# B&R Automation Studio project CoffeeMachine
Automation Studio 4.12.9.18 SP; Default project; technology packages: Acp10Arnc0 5.16.2

## Configuration PP65mcSim

CPU 4PP065.0571-P74, AutomationRuntime E3.10, Build 4.1.2, Safety 0.0, Vc V4.72.6

### Task classes (Cpu.sw)
```
Cyclic#1 (cycle 10000 us, tolerance 10000 us):
  mainlogic <- mainlogic.prg
  feeder <- FeederArm.feeder.prg
  conveyor <- ConveyorBelt.conveyor.prg
  brewing <- BrewingAssembly.brewing.prg
  heating <- FlowHeater.heating.prg
Cyclic#4 (cycle 100000 us, tolerance 100000 us):
  visCtrl <- Visualisation.visCtrl.prg
  visAlarm <- Visualisation.visAlarm.prg
  visTrend <- Visualisation.visTrend.prg
DataObjects: cappu <- Recipes.cappu.dob, regular <- Recipes.regular.dob, espres <- Recipes.espres.dob, Acp10sys
NcDataObjects: acp_err <- FeederArm.acp_err.dob, motor_sim <- FeederArm.motor_sim.dob, motor_offi <- FeederArm.motor_office.dob, feed_ini <- FeederArm.feed_ini.dob, conv_ini <- ConveyorBelt.conv_ini.dob
Binaries: vccalarm, vcclbox, vcctext, vcrt, VisuW03, vccnum, vcchspot, vccbar, vccurl, vcchtml, vcfile, arialxsr, vcpdsw, vccbmp, vcshared, vcctrend, vcfntttf, vcgclass, vccovl, arialbd, vcdsint, vccslider, vcalarm, vccline, vcresman, vcdsloc, vccbtn, vccstr, vcbclass, vcxml, VisuW02, arial, vccdt, vccgauge, vccshape, arconfig, sysconf, ashwd, asfw, iomap, Acp10map, Acp10cfg, vctcal, vcpfmtcx, vcpdi815, VisuW01, visvc, vcpdi855, vcpfpp50, vcpdihd, vcptelo, vcmgr
Libraries: Acp10sdc, standard, loopconr, astime, runtime, powerlnk, CoffeeLib, Acp10par, AsArSdm, NcGlobal, brsystem, sys_lib, Acp10man, fileio, dataobj, acp10_mc, visapi
```

### Hardware
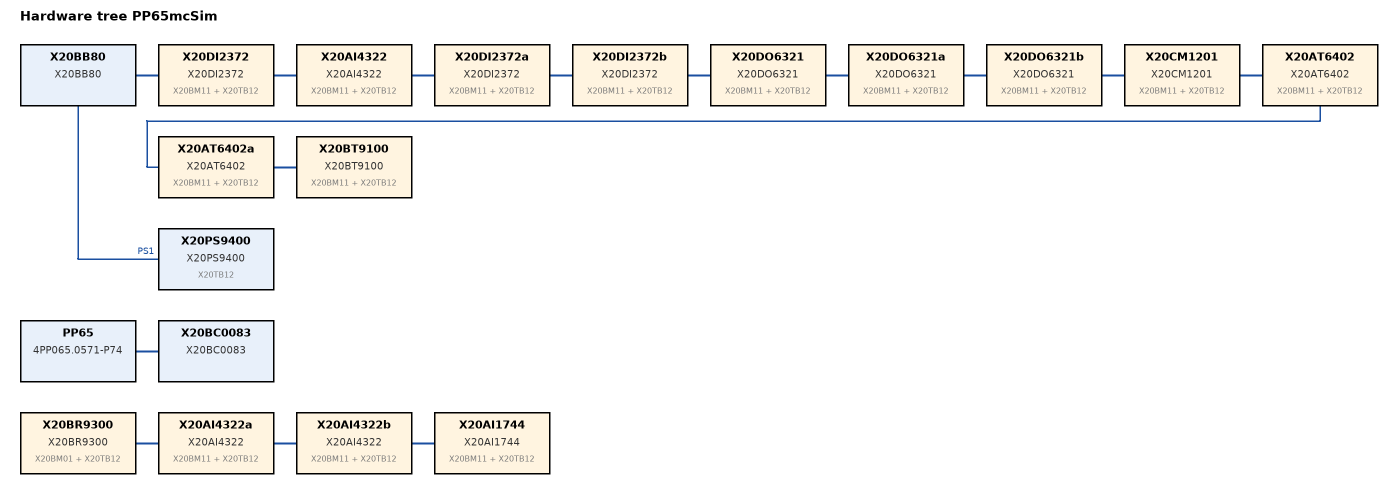
```
PP65 : 4PP065.0571-P74 v1.2.0.0
  Connector IF4:
    DNAConfiguration = manual
  Connector IF5:
    ActivateDevice = 1
    HostName = pp500coffeemachine
    Mode = Manual
    InternetAddress = 10.49.40.222
    SubnetMask = 255.255.255.0
  PreserveNonVolatileSystemSettings = 0
  BRObjects = 450
  Cyclic1Duration = 10000
  Cyclic1Tolerance = 10000
  Cyclic2Duration = 20000
  Cyclic2Tolerance = 20000
  Cyclic3Duration = 50000
  Cyclic3Tolerance = 50000
  Cyclic4Duration = 100000
  Cyclic4Tolerance = 100000
  Cyclic5Duration = 200000
  Cyclic5Tolerance = 200000
  Cyclic6Duration = 500000
  Cyclic6Tolerance = 500000
  Cyclic7Duration = 1000000
  Cyclic7Tolerance = 1000000
  Cyclic8Duration = 10000
  Cyclic8Tolerance = 30000000
  EthernetHostName = brautomation
  ActivateDns = 1
X20AI1744 : X20AI1744 v1.10.0.0  [SS1 -> X20TB12o.SS; SL -> X20BM11m.SL1]
  Supervision = off
X20AI4322 : X20AI4322 v1.2.0.0  [SS1 -> X20TB12b.SS; SL -> X20BM11a.SL1]
  Supervision = off
X20AI4322a : X20AI4322 v1.2.0.0  [SS1 -> X20TB12m.SS; SL -> X20BM11k.SL1]
  Supervision = off
X20AI4322b : X20AI4322 v1.2.0.0  [SS1 -> X20TB12n.SS; SL -> X20BM11l.SL1]
  Supervision = off
X20AT6402 : X20AT6402 v1.2.0.0  [SS1 -> X20TB12i.SS; SL -> X20BM11h.SL1]
  Supervision = off
X20AT6402a : X20AT6402 v1.2.0.0  [SS1 -> X20TB12j.SS; SL -> X20BM11i.SL1]
  Supervision = off
X20BB80 : X20BB80 v1.1.0.0
X20BC0083 : X20BC0083 v2.16.0.0  [PLK1 -> PP65.IF4 (NodeNumber=1) [Cable Type=PowerlinkCable, Length=10, Version=1.0.0.3]; SL -> X20BB80.SL1]
  Supervision = off
X20BM01 : X20BM01 v2.2.0.0
X20BM11 : X20BM11 v1.1.0.0  [X2X1 -> X20BB80.IF1]
X20BM11a : X20BM11 v1.1.0.0  [X2X1 -> X20BM11.X2X2]
X20BM11b : X20BM11 v1.1.0.0  [X2X1 -> X20BM11a.X2X2]
X20BM11c : X20BM11 v1.1.0.0  [X2X1 -> X20BM11b.X2X2]
X20BM11d : X20BM11 v1.1.0.0  [X2X1 -> X20BM11c.X2X2]
X20BM11e : X20BM11 v1.1.0.0  [X2X1 -> X20BM11d.X2X2]
X20BM11f : X20BM11 v1.1.0.0  [X2X1 -> X20BM11e.X2X2]
X20BM11g : X20BM11 v1.1.0.0  [X2X1 -> X20BM11f.X2X2]
X20BM11h : X20BM11 v1.1.0.0  [X2X1 -> X20BM11g.X2X2]
X20BM11i : X20BM11 v1.1.0.0  [X2X1 -> X20BM11h.X2X2]
X20BM11j : X20BM11 v1.1.0.0  [X2X1 -> X20BM11i.X2X2]
X20BM11k : X20BM11 v1.1.0.0  [X2X1 -> X20BM01.X2X2]
X20BM11l : X20BM11 v1.1.0.0  [X2X1 -> X20BM11k.X2X2]
X20BM11m : X20BM11 v1.1.0.0  [X2X1 -> X20BM11l.X2X2]
X20BR9300 : X20BR9300 v1.3.0.0  [SS1 -> X20TB12l.SS; SL -> X20BM01.SL1; X2X1 -> X20BT9100.X2X1 [Cable Type=X2XCable, Length=10, Version=1.0.0.3]]
  Supervision = off
X20BT9100 : X20BT9100 v1.3.0.0  [SS1 -> X20TB12k.SS; SL -> X20BM11j.SL1]
  Supervision = off
X20CM1201 : X20CM1201 v1.2.0.0  [SS1 -> X20TB12h.SS; SL -> X20BM11g.SL1]
  Supervision = off
X20DI2372 : X20DI2372 v1.2.0.0  [SS1 -> X20TB12a.SS; SL -> X20BM11.SL1]
  Supervision = off
X20DI2372a : X20DI2372 v1.2.0.0  [SS1 -> X20TB12c.SS; SL -> X20BM11b.SL1]
  Supervision = off
X20DI2372b : X20DI2372 v1.2.0.0  [SS1 -> X20TB12d.SS; SL -> X20BM11c.SL1]
  Supervision = off
X20DO6321 : X20DO6321 v1.2.0.0  [SS1 -> X20TB12e.SS; SL -> X20BM11d.SL1]
  Supervision = off
X20DO6321a : X20DO6321 v1.2.0.0  [SS1 -> X20TB12f.SS; SL -> X20BM11e.SL1]
  Supervision = off
X20DO6321b : X20DO6321 v1.2.0.0  [SS1 -> X20TB12g.SS; SL -> X20BM11f.SL1]
  Supervision = off
X20PS9400 : X20PS9400 v1.8.0.0  [SS1 -> X20TB12.SS; PS -> X20BB80.PS1]
  Supervision = off
X20TB12 : X20TB12 v1.0.0.0
X20TB12a : X20TB12 v1.0.0.0
X20TB12b : X20TB12 v1.0.0.0
X20TB12c : X20TB12 v1.0.0.0
X20TB12d : X20TB12 v1.0.0.0
X20TB12e : X20TB12 v1.0.0.0
X20TB12f : X20TB12 v1.0.0.0
X20TB12g : X20TB12 v1.0.0.0
X20TB12h : X20TB12 v1.0.0.0
X20TB12i : X20TB12 v1.0.0.0
X20TB12j : X20TB12 v1.0.0.0
X20TB12k : X20TB12 v1.0.0.0
X20TB12l : X20TB12 v1.0.0.0
X20TB12m : X20TB12 v1.0.0.0
X20TB12n : X20TB12 v1.0.0.0
X20TB12o : X20TB12 v1.0.0.0
```

## Configuration Simulation

CPU , AutomationRuntime I4.93, Build 4.1.2, Safety 0.0, Vc V4.73.3

### Task classes (AppMo.sw)
```
Cyclic#1 (cycle 10000 us, tolerance 0 us):
  myApptask1 <- myAppMod1.myApptask1.prg
```

### Task classes (Cpu.sw)
```
Cyclic#1 (cycle 10000 us, tolerance 0 us):
  mainlogic <- mainlogic.prg
  feeder <- FeederArm.feeder.prg
  conveyor <- ConveyorBelt.conveyor.prg
  brewing <- BrewingAssembly.brewing.prg
  heating <- FlowHeater.heating.prg
Cyclic#2:
  visCtrl <- Visualisation.visCtrl.prg
Cyclic#4:
  visAlarm <- Visualisation.visAlarm.prg
  visTrend <- Visualisation.visTrend.prg
  myProg <- myProg.prg
DataObjects: regular <- Recipes.regular.dob, cappu <- Recipes.cappu.dob, espres <- Recipes.espres.dob, empty1 <- Recipes.empty1.dob, object2 <- Recipes.object2.dob, data <- data.dob
NcDataObjects: acp_err <- FeederArm.acp_err.dob, motor_sim <- FeederArm.motor_sim.dob, motor_offi <- FeederArm.motor_office.dob, feed_ini <- FeederArm.feed_ini.dob, conv_ini <- ConveyorBelt.conv_ini.dob, cnc1 <- cnc1.dob, cnc2 <- cnc2.dob, cnc3 <- cnc3.dob
VcDataObjects: Visu <- Visualisation.Visu.dob
Binaries: vccslider, vccurl, vcxml, vcchtml, arialxsr, vcchspot, vcctext, vcresman, vccovl, vcfile, vcdsloc, vcbclass, vcfntttf, vccstr, vcgclass, vcshared, vcrt, vccbmp, vccbar, vccbtn, vcmgr, vctcal, visvc, vcalarm, vccnum, vcdsint, vccalarm, vccline, vcpdvnc, vcpdsw, vcnet, vcctrend, vcclbox, vcpfar00, Visu01, Visu02, Visu03, vccgauge, vccshape, vccdt, ARIALBD, ARIAL, Acp10cfg, Acp10map, iomap, sysconf, ashwd, asfw, arconfig, ARIALU_1, vcbmpng, arialu_1, acp10map, acp10cfg, arialbd, arial
Libraries: AsTime, CoffeeLib, FileIO, NcGlobal, Acp10par, Convert, Visapi, AsArSdm, Runtime, operator, standard, dataobj, powerlnk, brsystem, sys_lib, Acp10man, Acp10sim, Acp10_MC, Acp10sdc, AsArProf, loopconr, vcscrsht
```

### Hardware
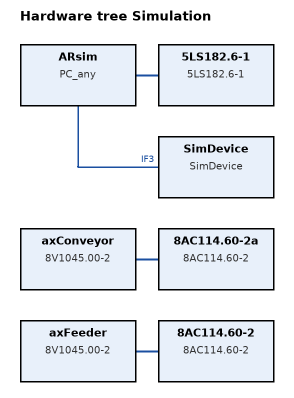
```
5LS182.6-1 : 5LS182.6-1 v1.5.0.0  [SL -> ARsim.SL1]
  Connector IF1:
    DNAConfiguration = manual
8AC114.60-2 : 8AC114.60-2 v1.0.0.8  [SS -> axFeeder.SS1; PLK1 -> 5LS182.6-1.IF1 (NodeNumber=1) [Cable Type=PowerlinkCable, Length=10, Version=1.0.0.3]; PLK2 -> 8AC114.60-2a.PLK1 (NodeNumber=1) [Cable Type=PowerlinkCable, Length=10, Version=1.0.0.3]]
8AC114.60-2a : 8AC114.60-2 v1.0.0.8  [SS -> axConveyor.SS1; PLK1 -> 8AC114.60-2.PLK2 (NodeNumber=2) [Cable Type=PowerlinkCable, Length=10, Version=1.0.0.3]]
ARsim : PC_any v1.1.1.0 (OrderNumber=PC)
  Connector IF3:
    Vnc1
    VncVcObjectName1 = Visu
    VncAuthentication1 = 1
    VncPasswordViewOnly1 = v
    VncPasswordViewControl1 = c
    VncRefreshRate1 = 200
    VncTitle1 = VNC - B&R Coffee Machine
  ConfigurationID = CoffeeMachine_Simulation
  XLinkUseDefault = 0
  Cyclic1Duration = 10000
  Cyclic1Tolerance = 0
  FileDevice1
  FileDeviceName1 = USER
  FileDevicePath1 = USER_PATH
  ActivateOpcUa = 1
  OpcUaInformationModels_PV_Version = 1
SimDevice : SimDevice v1.0.0.5  [ETH1 -> ARsim.IF3 [Cable Type=PowerlinkCable, Length=10, Version=1.0.0.3]]
  Channel1
  ChannelID1 = input
  ChannelDirection1 = IN
  Channel2
  ChannelID2 = output
axConveyor : 8V1045.00-2 v2.2.0.0
  Simulate = standard
axFeeder : 8V1045.00-2 v2.2.0.0
  Simulate = standard
```

### IoMap.iom - ARsim/IoMap.iom
```iecst
(********************************************************************
 * COPYRIGHT -- B&R
 ********************************************************************
 * File: IoMap.iom
 * Author: B&R
 * Created: June 06, 2007
 ********************************************************************
 * IO mapping file
 ********************************************************************)
VAR_CONFIG
	Cyclic#4.::diStartCoffee AT %IX."SimDevice".input;
	Cyclic#4.::doCupPull AT %QX."SimDevice".output;
END_VAR
```

### Acp10map.ncm - ARsim/Motion/Acp10map.ncm
```
NcMapping (NcSwId=acp10)
  NcObject axFeeder (ModuleId=axFeeder, Type=ncAXIS, Channel=1, AcoposSimulation=Standard, InitParameter=feed_ini, AcoposParameter=motor_sim, AdditionalData=PLCopen_ModPos="36000,100", Disabled=FALSE, ModuleDisabled=FALSE)
  NcObject axConveyor (ModuleId=axConveyor, Type=ncAXIS, Channel=1, AcoposSimulation=Standard, InitParameter=conv_ini, AcoposParameter=motor_sim, AdditionalData=PLCopen_ModPos="8388608,100", Disabled=FALSE, ModuleDisabled=FALSE)
```

## Logical view

Binary libraries used (declarations not repeated): Convert, Runtime, sys_lib, brsystem, Standard, AsString, DataObj, FileIO, operator, AsTime, Visapi, AsArSdm, AsArProf, LoopConR 4.10.2, Acp10man 5.16.2, Acp10par 5.16.2, NcGlobal 5.16.2, Acp10sdc 5.16.2, Acp10sim 5.16.2, Acp10_MC 5.16.2

### Package Logical/Doc - Project Documentation

### Global.typ - Global Data Types
```iecst
(********************************************************************
 * COPYRIGHT -- B&R
 ********************************************************************
 * File: Global.typ
 * Author: B&R
 * Created: June 06, 2007
 ********************************************************************
 * Global data types of project coffee
 ********************************************************************)

TYPE
	feeder_status_typ : 	STRUCT
		power : BOOL;
		home : BOOL;
		axisErrorNumber : UINT;
		axisErrorText : STRING[255];
	END_STRUCT;
	feeder_cmd_typ : 	STRUCT
		requestToPut : BOOL;
	END_STRUCT;
	feeder_typ : 	STRUCT
		cmd : feeder_cmd_typ;
		status : feeder_status_typ;
	END_STRUCT;
	main_status_money_typ : 	STRUCT
		changedMoney : REAL;
		cent1 : USINT;
		cent2 : USINT;
		cent5 : USINT;
		cent10 : USINT;
		cent20 : USINT;
		cent50 : USINT;
		euro1 : UDINT;
		euro2 : UDINT;
	END_STRUCT;
	main_status_progress_typ : 	STRUCT
		total : REAL;
		current : REAL;
	END_STRUCT;
	main_status_typ : 	STRUCT
		money : main_status_money_typ;
		progressStep : USINT;
		curPage : UINT;
		curLanguage : UINT;
		startProgressStep : USINT;
	END_STRUCT;
	main_par_recipe_typ : 	STRUCT
		price : REAL;
		setTemp : REAL;
		milk : REAL;
		sugar : REAL;
		coffee : REAL;
		water : REAL;
	END_STRUCT;
	main_par_typ : 	STRUCT
		coffeeType : SINT;
		givenMoney : REAL;
		recipe : main_par_recipe_typ;
	END_STRUCT;
	main_cmd_typ : 	STRUCT
		switchOnOff : BOOL;
		errorAck : BOOL;
		start : BOOL;
		vis : main_cmd_vis_typ;
	END_STRUCT;
	main_cmd_vis_typ : 	STRUCT
		newPage : UINT;
		startFlag : BOOL;
		startButtonColor : UINT;
		waterTempColor : UINT;
		messageColor : UINT;
		messageIndex : USINT;
		euro2hidden : UINT;
		euro1hidden : UINT;
		cent50hidden : UINT;
		cent20hidden : UINT;
		cent10hidden : UINT;
		cent5hidden : UINT;
		cent2hidden : UINT;
		cent1hidden : UINT;
		newLanguage : UINT;
	END_STRUCT;
	main_typ : 	STRUCT
		cmd : main_cmd_typ;
		par : main_par_typ;
		status : main_status_typ;
	END_STRUCT;
	conveyor_typ : 	STRUCT
		status : conveyor_status_typ;
	END_STRUCT;
	conveyor_status_typ : 	STRUCT
		power : BOOL;
		home : BOOL;
		axisErrorNumber : UINT;
		axisErrorText : STRING[255];
		readyToTake : BOOL;
	END_STRUCT;
	brewing_par_typ : 	STRUCT
		coffeeType : USINT;
	END_STRUCT;
	brewing_cmd_typ : 	STRUCT
		start : BOOL;
	END_STRUCT;
	brewing_status_typ : 	STRUCT
		done : BOOL;
		sBrewingStep : UINT;
		brewingStepText : STRING[64];
	END_STRUCT;
	brewing_typ : 	STRUCT
		cmd : brewing_cmd_typ;
		par : brewing_par_typ;
		status : brewing_status_typ;
	END_STRUCT;
	heating_status_typ : 	STRUCT
		setTempOK : BOOL;
		actTemp : REAL;
	END_STRUCT;
	heating_cmd_typ : 	STRUCT
		start : BOOL;
		updatePIDpar : BOOL;
	END_STRUCT;
	heating_typ : 	STRUCT
		cmd : heating_cmd_typ;
		status : heating_status_typ;
	END_STRUCT;
END_TYPE
```

### Package Logical/ConveyorBelt - Conveyor Control

- Data object Logical/ConveyorBelt/conv_ini (Ax) (no source held here)

### conveyor.var
```iecst
(********************************************************************
 * COPYRIGHT -- B&R
 ********************************************************************
 * Package: conveyor
 * File: conveyor.var
 * Author: B&R
 * Created: June 14, 2007
 *******************************************************************)
VAR
	conveyorMC_Power : MC_Power;
	conveyorMC_Home : MC_Home;
	conveyorMC_ReadAxisError : MC_ReadAxisError;
	conveyorMC_Reset : MC_Reset;
	conveyorMC_MoveAdditive : MC_MoveAdditive;
	conveyorTakeoutMC_MoveAdditve : MC_MoveAdditive;
	conveyorMC_ReadStatus : MC_ReadStatus;
	MC_ReadActualPosition_0 : MC_ReadActualPosition;
	MC_ReadActualVelocity_0 : MC_ReadActualVelocity;
END_VAR
```

### Package Logical/BrewingAssembly - Brewing & Dosing

### Program Logical/BrewingAssembly/brewing (IEC) - Brewing Logic Control

#### brewing.st
```iecst
(********************************************************************
 * COPYRIGHT -- B&R
 ********************************************************************
 * Program: Brewing
 * File: Brewing.st
 * Author: B&R
 * Created: June 12, 2007
 ********************************************************************
 * Implementation of program Brewing
 ********************************************************************)

PROGRAM _CYCLIC
	(* plain text information of current step *)
	IF (pBrewingText <> 0) THEN
			strcpy(ADR(gBrewing.status.brewingStepText), pBrewingText);
	END_IF

	IF EDGEPOS(diStartCoffee) = TRUE THEN
 		gMainLogic.status.progressStep := 0;			(* transporting cup to brewing station *)
	END_IF

	CASE gBrewing.status.sBrewingStep OF
		(* wait for start signal *)
		sSTANDBY:
			pBrewingText := ADR('sSTANDBY');

			IF (gBrewing.cmd.start = TRUE) THEN
				gMainLogic.status.progressStep := 1;			(* brewing in progress *)
   			    gBrewing.cmd.start   := FALSE;
				gBrewing.status.done := FALSE;
				gBrewing.status.sBrewingStep := sDOSING;
			END_IF

		(* dose ingredients according to recipe *)
		sDOSING:
			pBrewingText := ADR('sDOSING');

			milkTP  (IN := 1, PT := REAL_TO_TIME(gMainLogic.par.recipe.milk   * 10));	(* 100ml -> 1s *)
			sugarTP (IN := 1, PT := REAL_TO_TIME(gMainLogic.par.recipe.sugar  * 10));  (* 50g -> 500ms *)
			coffeeTP(IN := 1, PT := REAL_TO_TIME(gMainLogic.par.recipe.coffee * 10));  (* 80g -> 800ms *)

			doDoseMilk   := milkTP.Q;
			doDoseSugar  := sugarTP.Q;
			doDoseCoffee := coffeeTP.Q;

			(* wait until dosing is finished *)
			IF (milkTP.Q = 0) AND (sugarTP.Q = 0) AND (coffeeTP.Q = 0) THEN
				milkTP  (IN := 0, PT := 0);
				sugarTP (IN := 0, PT := 0);
				coffeeTP(IN := 0, PT := 0);
	 			gBrewing.status.sBrewingStep := sBREWING;
	 		END_IF

		(* brew coffee *)
		sBREWING:
			pBrewingText := ADR('sBREWING');

			(* start brewing if set temperature has been reached *)
			IF (gHeating.status.setTempOK = TRUE) THEN
				waterTP(IN := 1, PT := REAL_TO_TIME(gMainLogic.par.recipe.water * 50));		(* 100ml -> 1s *)

				doPumpWater := waterTP.Q;

				(* wait until dosing is finished *)
				IF (waterTP.Q = 0) THEN
					waterTP(IN := 0, PT := 0);
		 			gBrewing.status.sBrewingStep := sFINISH;
		 		END_IF
			END_IF

		(* all done *)
		sFINISH:
			pBrewingText := ADR('sFINISH');

			gMainLogic.status.progressStep := 2;			(* ready for take out *)

			gBrewing.status.done := TRUE;
			gBrewing.status.sBrewingStep := sSTANDBY;
	END_CASE;
END_PROGRAM
```

### Package Logical/FeederArm - Feeder Control

### Data object Logical/FeederArm/motor_sim (Apt) - Parameters for motor simulation

#### motor_sim.apt
```
AcoposParameterTable:
  Root Parameters:
    110 = ncSW_ON (Name=CMD_SIMULATION)  // Simulation mode: Command
```

### Data object Logical/FeederArm/motor_office (Apt) - ACOPOS Parameter Table

#### motor_office.apt
```
AcoposParameterTable:
  Root Parameters:
    80 = 1 (Name=PHASE_MON_IGNORE)  // Power mains: Ignore phase failure
    390 = 24 (Name=UDC_NOMINAL, Unit=V)  // CTRL DC bus: Nominal voltage
```

### Data object Logical/FeederArm/feed_ini (Ax) - Feeder axis configuration

#### feed_ini.ax
```
InitParameter (Version=2.28.2, NcSwId=ACP10)
  ACP10AXIS_typ:
    dig_in:
      level:
        reference = ncACTIV_HI
        pos_hw_end = ncACTIV_HI
        neg_hw_end = ncACTIV_HI
        trigger1 = ncACTIV_HI
        trigger2 = ncACTIV_HI
    encoder_if:
      parameter:
        count_dir = ncSTANDARD
        scaling:
          load:
            units = 36000
            rev_motor = 10
    limit:
      parameter:
        v_pos = 10000
        v_neg = 10000
        a1_pos = 50000
        a2_pos = 50000
        a1_neg = 50000
        a2_neg = 50000
        t_jolt = 0.05
        t_in_pos = 0
        pos_sw_end = 8388607
        neg_sw_end = -8388608
        ds_warning = 500
        ds_stop = 1000
        a_stop = 1e+030
        dv_stop = 0
        dv_stop_mode = ncOFF
    controller:
      mode = ncPOSITION
      position:
        kv = 50
        tn = 0
        t_predict = 0.0008
        t_total = 0.0008
        p_max = 10000
        i_max = 0
      speed:
        kv = 2
        tn = 0
        t_filter = 0
        isq_filter1:
          type = ncOFF
          a0 = 0
          a1 = 0
          b0 = 0
          b1 = 0
          b2 = 0
          c0_par_id = 0
          c1_par_id = 0
        isq_filter2:
          type = ncOFF
          a0 = 0
          a1 = 0
          b0 = 0
          b1 = 0
          b2 = 0
          c0_par_id = 0
          c1_par_id = 0
        isq_filter3:
          type = ncOFF
          a0 = 0
          a1 = 0
          b0 = 0
          b1 = 0
          b2 = 0
          c0_par_id = 0
          c1_par_id = 0
      uf:
        type = ncLINEAR
        auto_config = ncMOTOR_PAR
        u0 = 0
        un = 0
        fn = 50
        k_f_slip = 0
      ff:
        torque_load = 0
        torque_pos = 0
        torque_neg = 0
        kv_torque = 0
        inertia = 0
        t_filter_a = 0
    move:
      stop:
        parameter[0]:
          decel_ramp = ncA_LIMIT
          controller = ncON
        parameter[1]:
          decel_ramp = ncA_LIMIT
          controller = ncON
        parameter[2]:
          decel_ramp = ncA_LIMIT
          controller = ncON
        parameter[3]:
          decel_ramp = ncA_LIMIT
          controller = ncON
        quickstop:
          decel_ramp = ncA_LIMIT
        drive_error:
          decel_ramp = ncA_LIMIT
      homing:
        parameter:
          s = 0
          v_switch = 5000
          v_trigger = 500
          a = 50000
          mode = ncDIRECT
          edge_sw = ncPOSITIVE
          start_dir = ncPOSITIVE
          trigg_dir = ncPOSITIVE
          ref_pulse = ncOFF
          tr_s_block = 0
      basis:
        parameter:
          v_pos = 10000
          v_neg = 10000
          a1_pos = 50000
          a2_pos = 50000
          a1_neg = 50000
          a2_neg = 50000
    message:
      text:
        parameter:
          format = ncBREAK
          columns = 80
          data_modul = acp_err
```

### Program Logical/FeederArm/feeder (IEC) - feeder logic control

#### feeder.var
```iecst
(********************************************************************
 * COPYRIGHT -- B&R
 ********************************************************************
 * Program: feeder
 * File: feeder.var
 * Author: B&R
 * Created: June 13, 2007
 ********************************************************************
 * Local variables of program feeder
 ********************************************************************)
VAR
	feederMC_Power : MC_Power;
	feederMC_Home : MC_Home;
	feederMC_ReadAxisError : MC_ReadAxisError;
	feederMC_Reset : MC_Reset;
	feederMC_MoveAdditive : MC_MoveAdditive;
	feederMC_ReadStatus : MC_ReadStatus;
	MC_ReadActualPosition_0 : MC_ReadActualPosition;
	MC_ReadActualVelocity_0 : MC_ReadActualVelocity;
END_VAR
```

### Package Logical/FlowHeater - Heater Control

### Program Logical/FlowHeater/heating (ANSIC) - Heating PID

#### heating.c
```c
/********************************************************************
 * COPYRIGHT -- B&R
 ********************************************************************
 * Program: Heating
 * File: Heating.c
 * Author: B&R
 * Created: June 12, 2007
 ********************************************************************
 * Implementation of program Heating
 ********************************************************************/

#include <bur/plctypes.h>

#ifdef _DEFAULT_INCLUDES
 #include <AsDefault.h>
#endif

/* prototyping */
BOOL inWindow(REAL set, REAL act, REAL window);

void _INIT HeatingINIT( void )
{
	/* PID parameters for water flow heater */
	tempLCRPIDpara.WX_max   = 100.0;
	tempLCRPIDpara.WX_min   = 0.0;
	tempLCRPIDpara.invert   = 0;
	tempLCRPIDpara.deadband = 0.0;
	tempLCRPIDpara.dY_max   = 0.0;
	tempLCRPIDpara.Kp       = 1.8; 		/*2.7;*/
	tempLCRPIDpara.Tn       = 12.0; 	/*6.2;*/
	tempLCRPIDpara.Tv       = 0.0; 		/*1.6;*/
	tempLCRPIDpara.Tf       = 0.0; 		/*0.16;*/
	tempLCRPIDpara.Kw       = 1.0;
	tempLCRPIDpara.Kfbk     = 1.0;		/* windup damping enabled */
	tempLCRPIDpara.fbk_mode = LCRPID_FBK_MODE_INTERN;
	tempLCRPIDpara.d_mode   = LCRPID_D_MODE_X;

	gHeating.cmd.updatePIDpar = 1;

	/* simulation of water pipe */
	simLCRPT2.V     = 3.9;
	simLCRPT2.T1    = 0.9;
	simLCRPT2.T2    = 15.3;
	simLCRPT2.y_set = 20.0;       		/* for simulation start at minimum controller output */
	simLCRPT2.set   = 1;

	/* Parameters for PID controller */
	tempLCRPID.Y_max  = 100.0;
	tempLCRPID.Y_min  = 20.0 / simLCRPT2.V;       /* limited to defined environmental temperature */
	tempLCRPID.A      = 0.0;
	tempLCRPID.Y_man  = 0.0;
	tempLCRPID.Y_fbk  = 0.0;
	tempLCRPID.hold_I = 0;
	tempLCRPID.mode   = LCRPID_MODE_CLOSE;

}

void _CYCLIC HeatingCYCLIC( void )
{
	/* update PID parameters */
	tempLCRPIDpara.enable = 1;
	tempLCRPIDpara.enter  = gHeating.cmd.updatePIDpar;
	LCRPIDpara(&tempLCRPIDpara);	/* LCRPIDpara function block call */

	gHeating.cmd.updatePIDpar = 0;

	/* start heating as soon as machine is switched on */
	tempLCRPID.enable = 1;
	if (gMainLogic.cmd.switchOnOff)
	{
		tempLCRPID.mode = LCRPID_MODE_AUTO;
	}
	else
	{
		tempLCRPID.mode = LCRPID_MODE_CLOSE;
	}
	tempLCRPID.ident  = tempLCRPIDpara.ident; /* ident of PIDpara -> provides parameters (Kp, Tn, Tv, ...) */
	tempLCRPID.W      = gMainLogic.par.recipe.setTemp;
	tempLCRPID.X      = gHeating.status.actTemp;
	LCRPID(&tempLCRPID);

	aoHeating = (INT)tempLCRPID.Y;

	/* PT2 element */
	simLCRPT2.enable  = 1;
	simLCRPT2.x = tempLCRPID.Y;
	LCRPT2(&simLCRPT2);
	simLCRPT2.set = 0;

	gHeating.status.actTemp = simLCRPT2.y;

	/* generate temperature OK flag if temperature is within a certain tolerance window */
	gHeating.status.setTempOK = inWindow(gMainLogic.par.recipe.setTemp, gHeating.status.actTemp, 1.0);
}

BOOL inWindow(REAL set, REAL act, REAL window)
{
	REAL delta = set - act;

	if (delta < 0) delta *= -1;

	if (delta < window)
	{
		return 1;
	}
	else
	{
		return 0;
	}
}
```

### Package Logical/Recipes - Coffee Recipes

- Data object Logical/Recipes/empty1 (Simple) (no source held here)

- Data object Logical/Recipes/object2 (Simple) (no source held here)

### Data object Logical/Recipes/regular (Simple)

- Visualisation Logical/Visualisation (not shown)

### Package Logical/Libraries - Global Libraries

### Library Logical/Libraries/CoffeeLib (IEC)

#### CoffeeLib.st
```iecst
(********************************************************************
 * COPYRIGHT -- B&R
 ********************************************************************
 * Library: CoffeeLib
 * File: CoffeeLib.st
 * Author: B&R
 * Created: June 18, 2007
 ********************************************************************
 * Implementation of library CoffeeLib
 ********************************************************************)

(*tempChanges given money based on euros*)
FUNCTION_BLOCK MoneyChanger
	IF (executeOld <> execute) AND (execute = TRUE) THEN
 		(* plausibility check: *)
		IF (given < price) THEN
			cent1 := 0;
			cent2 := 0;
			cent5 := 0;
			cent10 := 0;
			cent20 := 0;
			cent50 := 0;
			euro1  := 0;
			euro2  := 0;
			RETURN;
		END_IF

		(* calculate change *)
		change := given - price;

		(* trim to two floating point digits -> cents *)
		change := UDINT_TO_REAL(REAL_TO_UDINT(change * 100)) / 100;

		(* EURO *)
		euro2 := TRUNC(change) / 2;
		euro1 := TRUNC(change) MOD 2;

		(* CENTS *)
		centChange := REAL_TO_USINT((change - TRUNC(change)) * 100.0);	(* get digits after floating point in front of floating point (integer) *)
		cent50     := centChange / 50;
		centChange := centChange MOD 50;
		cent20     := centChange / 20;
		centChange := centChange MOD 20;
		cent10     := centChange / 10;
		centChange := centChange MOD 10;
		cent5      := centChange / 5;
		centChange := centChange MOD 5;
		cent2      := centChange / 2;
		centChange := centChange MOD 2;
		cent1      := centChange;

		resetMoney := 0;
	ELSE
		(* do not touch reset if not active *)
		resetMoney := given;
	END_IF

	executeOld := execute;
END_FUNCTION_BLOCK
```

### Program Logical/myProg (IEC) - Program

#### Type.typ - Local data types
```iecst
TYPE
	myStructType2 : 	STRUCT
		struct1 : myStructType;
		structList : ARRAY[0..2]OF myStructType;
	END_STRUCT;
	myStructType : 	STRUCT
		member1 : USINT := 3;
		member2 : ARRAY[0..2]OF USINT := [33,44,55];
	END_STRUCT;
	myEnumType :
		(
		eins,
		zwei,
		drei
		);
	myDerivedType1 :USINT(4..6) ;
	myDerivedType2 :ARRAY[3..6]OF USINT;
	myComplexStructType : 	STRUCT
		bool : BOOL;
		usint : USINT;
		uint : UINT;
		udint : UDINT;
		sint : SINT;
		int : INT;
		dint : DINT;
		real : REAL;
		lreal : LREAL;
		time : TIME;
		tod : TIME_OF_DAY;
		date : DATE;
		dt : DATE_AND_TIME;
		string : STRING[80];
		wstring : WSTRING[80];
		stringlist : ARRAY[1..10]OF STRING[40] := ['A','B','C','D','E','F','G','H','I','J'];
		wstringlist : ARRAY[1..10]OF WSTRING[40] := ["A","B","C","D","E","F","G","H","I","J"];
		vector : ARRAY[1..10]OF REAL;
		intvector : ARRAY[0..9]OF INT;
		matrix : ARRAY[0..9,0..3]OF REAL;
		myStruct0 : myStructType;
		myStruct1 : ARRAY[0..1]OF myStructType;
		myStruct2 : ARRAY[2..2]OF myStructType;
		myStruct3 : ARRAY[-1..1]OF myStructType;
		myStruct4 : ARRAY[0..2,0..3]OF myStructType;
		myStruct5 : ARRAY[0..2]OF myStructType2;
		myStruct6 : ARRAY[1..2,-1..1]OF myStructType2;
		myEnum : myEnumType;
		enumlist : ARRAY[0..4]OF myEnumType;
		subrange1 : SINT(-3..6) ;
		derived1 : myDerivedType1;
		derived2 : myDerivedType2;
		n : USINT := 99;
	END_STRUCT;
END_TYPE
```

#### myProg.st - Implementation code
```iecst
(********************************************************************
 * COPYRIGHT -- B&R Industrial Automation GmbH
 ********************************************************************
 * Program: myProg
 * File: myProg.st
 * Author: hilchenbachc
 * Created: November 22, 2022
 ********************************************************************
 * Implementation of program myProg
 ********************************************************************)

PROGRAM _INIT
	myComplexStruct.usint := 11;
	myComplexStruct.uint  := 12;
	myComplexStruct.udint := 13;
	myComplexStruct.sint := -11;
	myComplexStruct.int  := -12;
	myComplexStruct.dint := -13;
	myComplexStruct.real := 3.1415;
	myComplexStruct.lreal := 2 * myComplexStruct.real;
	myComplexStruct.string := 'The quick brown fox jumps over the lazy dog';
	myComplexStruct.wstring := "The quick brown fox jumps over the lazy dog";
	myComplexStruct.tod := TOD#23:39:59.999;
	myComplexStruct.time := T#23d_20h_31m_23s_648ms;
	myComplexStruct.date := D#2017-02-07;
	myComplexStruct.dt := DT#2016-02-07-06:28:15;

	FOR i := 0 TO 9 DO
		myComplexStruct.vector[i+1] := 200 + i;
		myComplexStruct.intvector[i] := 300+ i;
		FOR j := 0 TO 3 DO
			myComplexStruct.matrix[i,j] := 1000 + (10 * i + j);
		END_FOR
	END_FOR

	FOR i := -1 TO +1 DO
		myComplexStruct.myStruct3[i].member1 := INT_TO_USINT(5+i);
		myComplexStruct.myStruct3[i].member2[0] := INT_TO_USINT(10+i);
		myComplexStruct.myStruct3[i].member2[1] := INT_TO_USINT(20+i);
		myComplexStruct.myStruct3[i].member2[2] := INT_TO_USINT(30+i);
	END_FOR

	FOR i := 0 TO 2 DO
		FOR j := 0 TO 3 DO
			myComplexStruct.myStruct4[i,j].member1 := INT_TO_USINT(10 * i +j);
			myComplexStruct.myStruct4[i,j].member2[0] := INT_TO_USINT(20 * i +j);
			myComplexStruct.myStruct4[i,j].member2[1] := INT_TO_USINT(30 * i +j);
			myComplexStruct.myStruct4[i,j].member2[2] := INT_TO_USINT(40 * i +j);
		END_FOR
	END_FOR

	FOR n := 0 TO 2 DO
		FOR i := 0 TO 2 DO
			myComplexStruct.myStruct5[n].struct1.member1 := INT_TO_USINT(3 + i+n);
			FOR j := 0 TO 2 DO
				myComplexStruct.myStruct5[n].structList[i].member1 := INT_TO_USINT(10 + i + n);
				myComplexStruct.myStruct5[n].struct1.member2[j] := INT_TO_USINT(+j+i+n);
				myComplexStruct.myStruct5[n].structList[i].member2[j] := INT_TO_USINT((i+1)*10 + j);
			END_FOR
		END_FOR
	END_FOR

	myComplexStruct.myEnum := drei;
	myComplexStruct.enumlist[0] := eins;
	myComplexStruct.enumlist[1] := zwei;
	myComplexStruct.enumlist[2] := drei;
	myComplexStruct.enumlist[3] := eins;
	myComplexStruct.enumlist[4] := zwei;

	myComplexStruct.derived2[3] := 3;
	myComplexStruct.derived2[4] := 4;
	myComplexStruct.derived2[5] := 5;
	myComplexStruct.derived2[6] := 6;
	sizeof_myComplexStruct := SIZEOF(myComplexStruct);

END_PROGRAM

PROGRAM _CYCLIC

END_PROGRAM
```

#### myProg.var - Local variables
```iecst
(********************************************************************
 * COPYRIGHT -- B&R Industrial Automation GmbH
 ********************************************************************
 * Program: myProg
 * File: myProg.var
 * Author: hilchenbachc
 * Created: November 22, 2022
 ********************************************************************
 * Local variables of program myProg
 ********************************************************************)
VAR
	myComplexStruct : myComplexStructType;
	i : INT;
	j : INT;
	n : USINT := 0;
	sizeof_myComplexStruct : UDINT;
END_VAR
```

### Data object Logical/cnc1 (Cnc) - CNC Program

#### NewCncProg.cnc
```
(*******************************************************************)
( COPYRIGHT -- B&R Industrial Automation GmbH )
(*******************************************************************)
( CNC program: NewCncProg )
( File: NewCncProg.cnc )
( Author: hilchenbachc )
( Created: December 21, 2022 )
(*******************************************************************)
( CNC program file: NewCncProg.cnc )
(*******************************************************************)

%001 (NewCncProg)

( TODO: Add code here )

N999 M30
```

- Data object Logical/data (Simple) - Simple data object (no source held here)

### Program Logical/myAppMod1/myApptask1 (IEC)

#### Variables.var
```iecst
VAR
	i : USINT := 0;
END_VAR
```

#### Main.st
```iecst
PROGRAM _INIT
	(* Insert code here *)

END_PROGRAM

PROGRAM _CYCLIC
	i := i + 1;

END_PROGRAM

PROGRAM _EXIT
	(* Insert code here *)

END_PROGRAM
```

Listed in the project but not available here: Logical/Global.var, Logical/mainlogic, Logical/FeederArm/acp_err, Logical/cnc3, Logical/cnc2
